Staubli VAL3: dataReceiver.pgx

program dataReceiver()
  local num l_nMsgRecvState
  local num l_nStartTime
begin
  // Copyright (c) 2016, Ocado Technology - Robotics Research Team
  //
  // Licensed under the Apache License, Version 2.0 (the "License");
  // you may not use this file except in compliance with the License.
  // You may obtain a copy of the License at
  //
  //     http://www.apache.org/licenses/LICENSE-2.0
  //
  // Unless required by applicable law or agreed to in writing, software
  // distributed under the License is distributed on an "AS IS" BASIS,
  // WITHOUT WARRANTIES OR CONDITIONS OF ANY KIND, either express or implied.
  // See the License for the specific language governing permissions and
  // limitations under the License.



  // state machine at initial state
  // 0: receive header
  // 1: decode header
  // 2: receive body
  // 3: decode body
  // 4: push motion into buffer
  // 5: send ACK

  // Set variable constants to make sure they were not changed
  nReset=0
  nRecHeader=0
  nDecHeader=1
  nRecBody=2
  nDecBody=3
  nPushMotion=4
  nAck=5

  l_nMsgRecvState=nRecHeader
while (true)
    // usually for state machines a switch-case statement is a neat implementation
    // HOWEVER, at every iteration of while() this task is sequenced and only called
    // after whatever ms is was defined when created.
    // As a result, receiving one single message, pushing motion and sending ACK
    // would take 6 * task period using switch-case statement.
    // The desirable behaviour is to receive and decode a full message, push motion
    // into buffer and then send ACK to client WITHIN ONE ITERATION of while(),
    // hence the if statement sequence below
    l_nStartTime=clock()
    if (l_nMsgRecvState==nRecHeader)
      call recvMsgHeader(l_nMsgRecvState)
    endIf
    nHeaderTime=clock()-l_nStartTime
    if (l_nMsgRecvState==nDecHeader)
      call decodeMsgHeader(l_nMsgRecvState)
    endIf
    if (l_nMsgRecvState==nRecBody)
      call recvMsgBody(l_nMsgRecvState)
    endIf
    if (l_nMsgRecvState==nDecBody)
      call decodeMsgBody(l_nMsgRecvState)
    endIf
    if (l_nMsgRecvState==nPushMotion)
      call pushMotion(l_nMsgRecvState)
    endIf
    if (l_nMsgRecvState==nAck)
      call encodeAck()
      call sendAck(l_nMsgRecvState)
    endIf
    nElapsedTime=clock()-l_nStartTime-nHeaderTime

    // assert state machine is working OK
    if (l_nMsgRecvState<nRecHeader or l_nMsgRecvState>nAck)
      popUpMsg("Data reception state machine error")
    endIf

    // sequence task
    delay(0)


  endWhile
end
